Fanuc KAREL source: kf00049.KL

PROGRAM KF00049
%STACKSIZE=65535
%PRIORITY=65535
%NOLOCKGROUP
VAR
I : INTEGER
J : INTEGER
X : REAL
Y : REAL
B : BOOLEAN
C : BOOLEAN
TXT : STRING[80]
TXT2 : STRING[80]
AI : ARRAY[4] OF INTEGER
BI : ARRAY[4] OF INTEGER
P : XYZWPR
JP : JOINTPOS9
PF : POSITION
STATUS : INTEGER
-- UNRESOLVED DECLARATIONS (source type spelling not recovered)
-- V1 : TYPE_0x0013 (type_u16=0x0013)
-- V2 : TYPE_0x0013 (type_u16=0x0013)
BEGIN
I=2
-- UNRESOLVED_PC line 22 opcodes [21 40 41 41 42] marker_code=16
-- UNSAFE_SOURCE_IR line 23: J = 10
J=20
END KF00049
